{attribute 'qualified_only'}
VAR_GLOBAL CONSTANT
	sPlainStringTopic	: STRING(255)	:= 'Plain Temperatures';	// this the topic we will publish on for plain string data
	sJsonStringTopic	: STRING(255)	:= 'JSON Temperatures';		// this the topic we will publish on for JSON formatted string data
	sBrokerAddress		: STRING(255)	:= 'test.mosquitto.org';	// this is the address of the MQTT broker we are using
	uiBrokerPort 		: UINT			:= 1883;					// the TCP port for the MQQT broker
END_VAR

(* stored: Version 1.1.0.1, ProductVersion 3.1.4024.3
   GVL Setup_Parameters: Id {b77ffd8f-1144-4dfe-b199-2cc07d0c0754} *)
